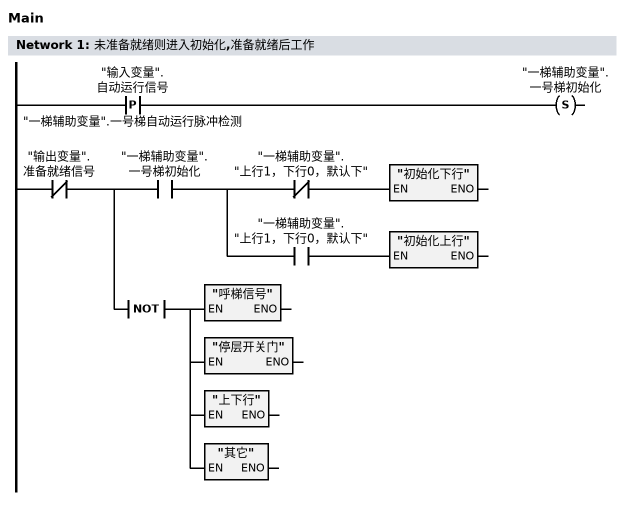
   RUNG wire#powerrail
      P_Contact(operand := "输入变量".自动运行信号, bit := "一梯辅助变量".一号梯自动运行脉冲检测)
      S_Coil( "一梯辅助变量".一号梯初始化 )
   END_RUNG
   RUNG wire#powerrail
      I_Contact( "输出变量".准备就绪信号 )
      wire#w1
      Contact( "一梯辅助变量".一号梯初始化 )
      wire#w2
      I_Contact( "一梯辅助变量"."上行1，下行0，默认下" )
      "初始化下行"()
   END_RUNG
   RUNG wire#w2
      Contact( "一梯辅助变量"."上行1，下行0，默认下" )
      "初始化上行"()
   END_RUNG
   RUNG wire#w1
      Not()
      wire#w3
      "呼梯信号"()
   END_RUNG
   RUNG wire#w3
      "停层开关门"()
   END_RUNG
   RUNG wire#w3
      "上下行"()
   END_RUNG
   RUNG wire#w3
      "其它"()
   END_RUNG
   // the same network as SCL:
   #_w1 := "输入变量".自动运行信号 AND NOT "一梯辅助变量".一号梯自动运行脉冲检测;   // rising edge of "输入变量".自动运行信号
   "一梯辅助变量".一号梯自动运行脉冲检测 := "输入变量".自动运行信号;
   IF #_w1 THEN "一梯辅助变量".一号梯初始化 := TRUE; END_IF;
   #_w2 := NOT "输出变量".准备就绪信号 AND "一梯辅助变量".一号梯初始化;
   #_w3 := NOT "输出变量".准备就绪信号;
   IF #_w2 AND NOT "一梯辅助变量"."上行1，下行0，默认下" THEN "初始化下行"(); END_IF;
   IF #_w2 AND "一梯辅助变量"."上行1，下行0，默认下" THEN "初始化上行"(); END_IF;
   IF NOT #_w3 THEN
       "呼梯信号"();
       "停层开关门"();
       "上下行"();
       "其它"();
   END_IF;
END_REGION
END_ORGANIZATION_BLOCK

(* ===== HMI "HMI_RT_1" =====
system functions are stored by id; their names below are inferred from use
connection "HMI_1": ETHERNET, S7_1500_OMS

HMI tags "默认变量表"
   "一梯辅助变量_1梯初始化到几层" : Int = PLC 一梯辅助变量.1梯初始化到几层 AT %DB29.DBW28, 1 s
   "一梯辅助变量_上行1，下行0，默认下" : Bool = PLC 一梯辅助变量.上行1，下行0，默认下 AT %DB29.DBX6.4, 1 s
   "输入变量_1号梯上端站第2限位" : Bool = PLC 输入变量.1号梯上端站第2限位 AT %DB1.DBX4.0, 1 s
   "输入变量_1号梯上端站第1限位" : Bool = PLC 输入变量.1号梯上端站第1限位 AT %DB1.DBX3.7, 1 s
   "一梯辅助变量_一号梯楼层数" : Int = PLC 一梯辅助变量.一号梯楼层数 AT %DB29.DBW4, 1 s
   "输入变量_1号梯下端站第1限位" : Bool = PLC 输入变量.1号梯下端站第1限位 AT %DB1.DBX4.1, 1 s
   "输入变量_1号梯下端站第2限位" : Bool = PLC 输入变量.1号梯下端站第2限位 AT %DB1.DBX4.2, 1 s
   "输出变量_1号梯满载指示" : Bool = PLC 输出变量.1号梯满载指示 AT %DB2.DBX3.4, 1 s
   "输出变量_1号梯下行指示" : Bool = PLC 输出变量.1号梯下行指示 AT %DB2.DBX3.0, 1 s
   "输出变量_1号梯上行指示" : Bool = PLC 输出变量.1号梯上行指示 AT %DB2.DBX2.7, 1 s
   "输出变量_准备就绪信号" : Bool = PLC 输出变量.准备就绪信号 AT %DB2.DBX4.7, 1 s
   "输出变量_1号梯LEDa" : Bool = PLC 输出变量.1号梯LEDa AT %DB2.DBX2.0, 1 s
   "输出变量_1号梯LEDb" : Bool = PLC 输出变量.1号梯LEDb AT %DB2.DBX2.1, 1 s
   "输出变量_1号梯LEDc" : Bool = PLC 输出变量.1号梯LEDc AT %DB2.DBX2.2, 1 s
   "输出变量_1号梯LEDd" : Bool = PLC 输出变量.1号梯LEDd AT %DB2.DBX2.3, 1 s
   "输出变量_1号梯LEDe" : Bool = PLC 输出变量.1号梯LEDe AT %DB2.DBX2.4, 1 s
   "输出变量_1号梯LEDf" : Bool = PLC 输出变量.1号梯LEDf AT %DB2.DBX2.5, 1 s
   "输出变量_1号梯LEDg" : Bool = PLC 输出变量.1号梯LEDg AT %DB2.DBX2.6, 1 s
   "输出变量_1号梯照明指示" : Bool = PLC 输出变量.1号梯照明指示 AT %DB2.DBX3.2, 1 s
   "输出变量_1号梯风扇指示" : Bool = PLC 输出变量.1号梯风扇指示 AT %DB2.DBX3.3, 1 s
   "输出变量_1号梯故障指示" : Bool = PLC 输出变量.1号梯故障指示 AT %DB2.DBX3.1, 1 s
   "一梯辅助变量_一层上呼标志" : Bool = PLC 一梯辅助变量.一层上呼标志 AT %DB29.DBX6.1, 1 s
   "一梯辅助变量_二层上呼标志" : Bool = PLC 一梯辅助变量.二层上呼标志 AT %DB29.DBX6.7, 1 s
   "一梯辅助变量_三层上呼标志" : Bool = PLC 一梯辅助变量.三层上呼标志 AT %DB29.DBX6.2, 1 s
   "一梯辅助变量_四层上呼标志" : Bool = PLC 一梯辅助变量.四层上呼标志 AT %DB29.DBX11.0, 1 s
   "一梯辅助变量_五层上呼标志" : Bool = PLC 一梯辅助变量.五层上呼标志 AT %DB29.DBX7.1, 1 s
   "一梯辅助变量_六层下呼标志" : Bool = PLC 一梯辅助变量.六层下呼标志 AT %DB29.DBX8.6, 1 s
   "一梯辅助变量_五层下呼标志" : Bool = PLC 一梯辅助变量.五层下呼标志 AT %DB29.DBX7.2, 1 s
   "一梯辅助变量_四层下呼标志" : Bool = PLC 一梯辅助变量.四层下呼标志 AT %DB29.DBX11.1, 1 s
   "一梯辅助变量_三层下呼标志" : Bool = PLC 一梯辅助变量.三层下呼标志 AT %DB29.DBX6.3, 1 s
   "一梯辅助变量_二层下呼标志" : Bool = PLC 一梯辅助变量.二层下呼标志 AT %DB29.DBX7.0, 1 s
   "一梯辅助变量_一号梯内选1" : Bool = PLC 一梯辅助变量.一号梯内选1 AT %DB29.DBX2.6, 1 s
   "一梯辅助变量_一号梯内选2" : Bool = PLC 一梯辅助变量.一号梯内选2 AT %DB29.DBX2.7, 1 s
   "一梯辅助变量_一号梯内选3" : Bool = PLC 一梯辅助变量.一号梯内选3 AT %DB29.DBX3.0, 1 s
   "一梯辅助变量_一号梯内选4" : Bool = PLC 一梯辅助变量.一号梯内选4 AT %DB29.DBX3.1, 1 s
   "一梯辅助变量_一号梯内选5" : Bool = PLC 一梯辅助变量.一号梯内选5 AT %DB29.DBX3.2, 1 s
   "一梯辅助变量_一号梯内选6" : Bool = PLC 一梯辅助变量.一号梯内选6 AT %DB29.DBX3.3, 1 s
   "一梯辅助变量_关门按钮标志" : Bool = PLC 一梯辅助变量.关门按钮标志 AT %DB29.DBX9.0, 1 s
   "一梯辅助变量_开门按钮标志" : Bool = PLC 一梯辅助变量.开门按钮标志 AT %DB29.DBX11.7, 1 s
   "输出变量_1号梯开门继电器" : Bool = PLC 输出变量.1号梯开门继电器 AT %DB2.DBX4.2, 1 s
   "输出变量_1号梯关门继电器" : Bool = PLC 输出变量.1号梯关门继电器 AT %DB2.DBX4.3, 1 s
   "输入变量_1号梯上平层信号" : Bool = PLC 输入变量.1号梯上平层信号 AT %DB1.DBX3.5, 1 s
   "输入变量_1号梯下平层信号" : Bool = PLC 输入变量.1号梯下平层信号 AT %DB1.DBX3.6, 1 s
   "输入变量_1号梯光幕信号" : Bool = PLC 输入变量.1号梯光幕信号 AT %DB1.DBX2.2, 1 s
   "输入变量_1号梯开门到位" : Bool = PLC 输入变量.1号梯开门到位 AT %DB1.DBX3.3, 1 s
   "输入变量_1号梯关门到位" : Bool = PLC 输入变量.1号梯关门到位 AT %DB1.DBX3.4, 1 s
   "输出变量_1号梯上行接触器" : Bool = PLC 输出变量.1号梯上行接触器 AT %DB2.DBX3.6, 1 s
   "输出变量_1号梯下行接触器" : Bool = PLC 输出变量.1号梯下行接触器 AT %DB2.DBX3.7, 1 s

text list "1号梯初始化楼层数": 1 '1层'; 2 '2层'; 3 '3层'; 4 '4层'; 5 '5层'; 6 '6层'

screen "1号梯" 1024x768
   TextField "文本域_37" at 51,288 size 150x31; Text '初始化控制'
   TextField "文本域_17" at 535,38 size 179x31; Text '运行信号指示'
   TextField "文本域_22" at 797,232 size 105x27; Text '故障指示'
   TextField "文本域_21" at 797,168 size 105x27; Text '轿内风扇'
   TextField "文本域_20" at 797,108 size 105x27; Text '轿内照明'
   TextField "文本域_18" at 541,83 size 105x27; Text '满载指示'
   Rectangle "矩形_8" at 688,96 size 64x14
      Appearance <- "输出变量_1号梯LEDa"
   Rectangle "矩形_9" at 751,110 size 13x65
      Appearance <- "输出变量_1号梯LEDb"
   Rectangle "矩形_10" at 677,110 size 13x65
      Appearance <- "输出变量_1号梯LEDf"
   Rectangle "矩形_11" at 690,175 size 64x14
      Appearance <- "输出变量_1号梯LEDg"
   Rectangle "矩形_12" at 752,187 size 13x65
      Appearance <- "输出变量_1号梯LEDc"
   Rectangle "矩形_13" at 678,187 size 13x65
      Appearance <- "输出变量_1号梯LEDe"
   Rectangle "矩形_14" at 690,252 size 64x14
      Appearance <- "输出变量_1号梯LEDd"
   TextField "文本域_19" at 541,172 size 105x27; Text '运行方向'
   Circle "圆_19" at 567,113 size 48x48
      Appearance <- "输出变量_1号梯满载指示"
   Circle "圆_20" at 915,95 size 48x48
      Appearance <- "输出变量_1号梯照明指示"
   Circle "圆_21" at 915,158 size 48x48
      Appearance <- "输出变量_1号梯风扇指示"
   Circle "圆_22" at 915,221 size 48x48
      Appearance <- "输出变量_1号梯故障指示"
   Polygon "多边形_5" at 572,205 size 37x59
      Appearance <- "输出变量_1号梯上行指示"
      Visibility <- "输出变量_1号梯上行指示"
   Polygon "多边形_7" at 573,207 size 37x59
      Appearance <- "输出变量_1号梯下行指示"
      Visibility <- "输出变量_1号梯下行指示"
   TextField "文本域_9" at 536,353 size 43x27; Text '1层'
   TextField "文本域_10" at 619,353 size 43x27; Text '2层'
   TextField "文本域_11" at 693,353 size 43x27; Text '3层'
   TextField "文本域_12" at 766,353 size 43x27; Text '4层'
   TextField "文本域_13" at 843,353 size 43x27; Text '5层'
   TextField "文本域_14" at 922,353 size 43x27; Text '6层'
   TextField "文本域_15" at 536,317 size 179x31; Text '厅外呼梯按钮'
   Group "Group_1" at 541,418 size 48x48
   Group "Group_2" at 619,390 size 48x48
   Group "Group_3" at 619,450 size 48x48
   Group "Group_4" at 693,390 size 48x48
   Group "Group_5" at 693,450 size 48x48
   Group "Group_6" at 765,390 size 48x48
   Group "Group_7" at 765,450 size 48x48
   Group "Group_8" at 843,390 size 48x48
   Group "Group_9" at 843,450 size 48x48
   Group "Group_10" at 919,418 size 48x48
   TextField "文本域_1" at 538,537 size 150x31; Text '轿厢内按钮'
   Group "Group_11" at 538,580 size 48x48
   Group "Group_12" at 610,580 size 48x48
   Group "Group_13" at 685,581 size 48x48
   Group "Group_14" at 759,580 size 48x48
   Group "Group_15" at 832,580 size 48x48
   Group "Group_16" at 911,581 size 48x48
   Group "Group_17" at 538,647 size 48x48
   Group "Group_18" at 610,647 size 48x48
   Rectangle "矩形_19" at 360,602 size 96x62
      Appearance <- "一梯辅助变量_一号梯楼层数"
   Rectangle "矩形_20" at 360,514 size 96x62
      Appearance <- "一梯辅助变量_一号梯楼层数"
   Rectangle "矩形_21" at 360,424 size 96x62
      Appearance <- "一梯辅助变量_一号梯楼层数"
   Rectangle "矩形_22" at 360,328 size 96x62
      Appearance <- "一梯辅助变量_一号梯楼层数"
   Rectangle "矩形_23" at 360,232 size 96x62
      Appearance <- "一梯辅助变量_一号梯楼层数"
   Rectangle "矩形_24" at 360,138 size 96x62
      Appearance <- "一梯辅助变量_一号梯楼层数"
   Rectangle "矩形_25" at 352,64 size 112x10
      Appearance <- "输入变量_1号梯上端站第2限位"
   Rectangle "矩形_26" at 352,86 size 112x10
      Appearance <- "输入变量_1号梯上端站第1限位"
   Rectangle "矩形_27" at 352,710 size 114x10
      Appearance <- "输入变量_1号梯下端站第2限位"
   Rectangle "矩形_28" at 352,690 size 112x10
      Appearance <- "输入变量_1号梯下端站第1限位"
   TextField "文本域_23" at 281,621 size 49x31; Text '1楼'
   TextField "文本域_24" at 281,530 size 49x31; Text '2楼'
   TextField "文本域_25" at 281,439 size 49x31; Text '3楼'
   TextField "文本域_26" at 281,348 size 49x31; Text '4楼'
   TextField "文本域_27" at 281,249 size 49x31; Text '5楼'
   TextField "文本域_28" at 281,150 size 49x31; Text '6楼'
   TextField "文本域_29" at 190,682 size 152x23; Text '下端站第一限位'
   TextField "文本域_30" at 190,704 size 152x23; Text '下端站第二限位'
   TextField "文本域_31" at 190,81 size 152x23; Text '上端站第一限位'
   TextField "文本域_32" at 190,58 size 152x23; Text '上端站第二限位'
   TextField "文本域_33" at 334,16 size 143x25; Text '电梯运行状态'
   TextField "文本域_34" at 46,124 size 150x31; Text '电梯门状态'
   TextField "文本域_35" at 46,166 size 121x31; Text '电梯开门'
   Rectangle "矩形_34" at 175,162 size 79x40
      Appearance <- "输出变量_1号梯开门继电器"
   TextField "文本域_36" at 46,220 size 121x31; Text '电梯关门'
   Rectangle "矩形_35" at 175,214 size 81x40
      Appearance <- "输出变量_1号梯关门继电器"
   SymbolicIOField "符号 I/O 域_1" at 153,344 size 109x45; TextOn '1'; TextOff '0'; TextList "1号梯初始化楼层数"
      ProcessValue <- "一梯辅助变量_1梯初始化到几层"
   TextField "文本域_39" at 156,391 size 92x31; Text '楼层数'
   Switch "Toggle_Vertical_G" at 54,334 size 83x97; CaptionText 'Switch'; TextOff '0'; TextOn '1'; PictureOff "Toggle_Vertical_G_Off_256c"; PictureOn "Toggle_Vertical_G_On_256c"
      on SwitchOff: ResetBit("一梯辅助变量_上行1，下行0，默认下")
      on SwitchOn: SetBit("一梯辅助变量_上行1，下行0，默认下")
   TextField "文本域_38" at 46,431 size 92x31; Text '上下行'
   Button "按钮_1" at 47,685 size 118x42; TextOff '返回登陆界面'
      on Click: ActivateScreen("登陆界面", 1)
   TextField "文本域_40" at 56,492 size 120x25; Text '上平层信号'
   Rectangle "矩形_39" at 176,486 size 62x30
      Appearance <- "输入变量_1号梯上平层信号"
   TextField "文本域_41" at 56,529 size 120x25; Text '下平层信号'
   Rectangle "矩形_41" at 176,523 size 62x30
      Appearance <- "输入变量_1号梯下平层信号"
   TextField "文本域_42" at 56,567 size 97x25; Text '光幕信号'
   Rectangle "矩形_43" at 176,561 size 62x30
      Appearance <- "输入变量_1号梯光幕信号"
   TextField "文本域_43" at 57,604 size 97x25; Text '开门到位'
   Rectangle "矩形_45" at 177,598 size 62x30
      Appearance <- "输入变量_1号梯开门到位"
   TextField "文本域_44" at 58,643 size 97x25; Text '关门到位'
   Rectangle "矩形_47" at 178,637 size 62x30
      Appearance <- "输入变量_1号梯关门到位"
   Group "Group" at 723,41 size 71x29
   Group "Group_19" at 699,538 size 71x29
   TextField "文本域_46" at 41,44 size 100x21; Text '下行接触器'
   Rectangle "矩形_52" at 143,39 size 45x30
      Appearance <- "输出变量_1号梯下行接触器"
   TextField "文本域_45" at 44,78 size 100x21; Text '上行接触器'
   Rectangle "矩形_50" at 143,73 size 45x30
      Appearance <- "输出变量_1号梯上行接触器"
   TextField "文本域_16" at 725,41 size 68x27; Text '1号梯'
      Appearance <- "输出变量_准备就绪信号"
   Rectangle "矩形_5" at 723,41 size 71x29
      Appearance <- "输出变量_准备就绪信号"
   Circle "圆_13" at 541,418 size 48x48
      Appearance <- "一梯辅助变量_一层上呼标志"
   Circle "圆_12" at 619,390 size 48x48
      Appearance <- "一梯辅助变量_二层上呼标志"
   Circle "圆_18" at 619,450 size 48x48
      Appearance <- "一梯辅助变量_二层下呼标志"
   Circle "圆_11" at 693,390 size 48x48
      Appearance <- "一梯辅助变量_三层上呼标志"
   Circle "圆_17" at 693,450 size 48x48
      Appearance <- "一梯辅助变量_三层下呼标志"
   Circle "圆_10" at 765,390 size 48x48
      Appearance <- "一梯辅助变量_四层上呼标志"
   Circle "圆_16" at 765,450 size 48x48
      Appearance <- "一梯辅助变量_四层下呼标志"
   Circle "圆_9" at 843,390 size 48x48
      Appearance <- "一梯辅助变量_五层上呼标志"
   Circle "圆_15" at 843,450 size 48x48
      Appearance <- "一梯辅助变量_五层下呼标志"
   Circle "圆_14" at 919,418 size 48x48
      Appearance <- "一梯辅助变量_六层下呼标志"
   Circle "圆_5" at 538,580 size 48x48
      Appearance <- "一梯辅助变量_一号梯内选1"
   TextField "文本域_2" at 551,589 size 20x31; Text '1'
   Circle "圆_4" at 610,580 size 48x48
      Appearance <- "一梯辅助变量_一号梯内选2"
   TextField "文本域_3" at 622,588 size 20x31; Text '2'
   Circle "圆_3" at 685,581 size 48x48
      Appearance <- "一梯辅助变量_一号梯内选3"
   TextField "文本域_4" at 699,589 size 20x31; Text '3'
   Circle "圆_2" at 759,580 size 48x48
      Appearance <- "一梯辅助变量_一号梯内选4"
   TextField "文本域_5" at 772,588 size 20x31; Text '4'
   Circle "圆_1" at 832,580 size 48x48
      Appearance <- "一梯辅助变量_一号梯内选5"
   TextField "文本域_6" at 845,587 size 20x31; Text '5'
   Circle "圆_6" at 911,581 size 48x48
      Appearance <- "一梯辅助变量_一号梯内选6"
   TextField "文本域_7" at 925,588 size 20x31; Text '6'
   Circle "圆_7" at 538,647 size 48x48
      Appearance <- "一梯辅助变量_开门按钮标志"
   Polygon "多边形_3" at 566,659 size 12x23
      Appearance <- "一梯辅助变量_开门按钮标志"
   Polygon "多边形_4" at 544,658 size 12x24
      Appearance <- "一梯辅助变量_开门按钮标志"
   Circle "圆_8" at 610,647 size 48x48
      Appearance <- "一梯辅助变量_关门按钮标志"
   Polygon "多边形_1" at 619,658 size 12x23
      Appearance <- "一梯辅助变量_关门按钮标志"
   Polygon "多边形_2" at 636,658 size 12x24
      Appearance <- "一梯辅助变量_关门按钮标志"
   TextField "文本域_8" at 701,538 size 68x27; Text '1号梯'
      Appearance <- "输出变量_准备就绪信号"
   Rectangle "矩形_3" at 699,538 size 71x29
      Appearance <- "输出变量_准备就绪信号"

screen "登陆界面" 1024x768
   Button "按钮_1" at 132,625 size 170x64; TextOff '返回监控画面'
      on Click: ActivateScreen("1号梯", 2)
*)